// Mitsubishi GX Works2 project: z10   PLC: Q02/Q02H

PROGRAM MAIN
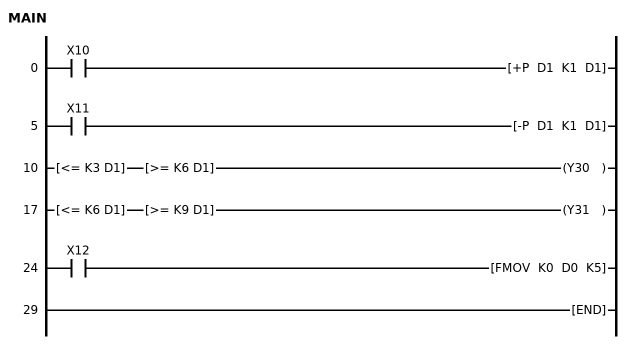
0     LD      X10
      +P      D1 K1 D1
5     LD      X11
      -P      D1 K1 D1
10    LD<=    K3 D1
      AND>=   K6 D1
      OUT     Y30
17    LD<=    K6 D1
      AND>=   K9 D1
      OUT     Y31
24    LD      X12
      FMOV    K0 D0 K5
29    END
END_PROGRAM
